FUNCTION_BLOCK InternalVariables (* Template for an empty basic function block *)
  (* Standard: 61499-2; Description: Copyright (c) 2019 Jan Holzweber This program and the accompanying materials are made available under the terms of the Eclipse Public License 2.0 which is available at https://www.eclipse.org/legal/epl-2.0/ SPDX-License-Identifier: EPL-2.0 *)
  (* Version 1.0, 2019-06-10, Jan Holzweber *)
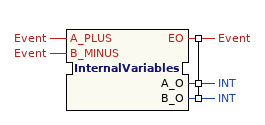
  EVENT_INPUT
    A_PLUS;
    B_MINUS;
  END_EVENT
  EVENT_OUTPUT
    EO WITH A_O, B_O;
  END_EVENT
  VAR_OUTPUT
    A_O : INT;
    B_O : INT;
  END_VAR
  VAR
    A : INT := 0; (* Internal Variable *)
    B : INT := 0; (* Internal Variable *)
  END_VAR
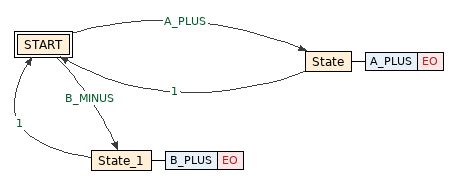
  EC_STATES
    START; (* Initial State *)
    State : A_PLUS -> EO;
    State_1 : B_PLUS -> EO;
  END_STATES
  EC_TRANSITIONS
    START TO State := A_PLUS;
    State TO START := 1;
    State_1 TO START := 1;
    START TO State_1 := B_MINUS;
  END_TRANSITIONS
  ALGORITHM A_PLUS IN ST: (* new algorithm *)
A_O:=A;
A:=A+1;
  END_ALGORITHM
  ALGORITHM B_PLUS IN ST: (* new algorithm *)
B_O:=B;
B:=B-1;
  END_ALGORITHM
END_FUNCTION_BLOCK
